Yaskawa INFORM job: FOLLOWBK.JBI

/JOB
//NAME FOLLOWBK
//POS
///NPOS 28,0,0,0,0,0
///TOOL 0
///POSTYPE PULSE
///PULSE
C00000=-2822,58859,-1118,-1041,-34109,-89
C00001=-2249,58669,-233,-1120,-33963,-317
C00002=-2249,58669,-1433,-1120,-33963,-317
C00003=-2021,58782,-1257,-1148,-34034,-410
C00004=-1683,58761,-1281,-1192,-34024,-546
C00005=-1595,58655,-1440,-1205,-33960,-580
C00006=-1505,58624,-1485,-1218,-33941,-615
C00007=-1505,58624,-285,-1218,-33941,-615
C00008=-1214,58456,-535,-1259,-33840,-730
C00009=-1214,58456,-1735,-1259,-33840,-730
C00010=-1059,58246,-2052,-1283,-33711,-789
C00011=-1059,58246,-852,-1283,-33711,-789
C00012=-2879,57741,-1646,-1051,-33397,-52
C00013=-2879,57741,-2846,-1051,-33397,-52
C00014=-2884,57537,-3152,-1053,-33275,-48
C00015=-2884,57537,-1952,-1053,-33275,-48
C00016=-2014,56709,-3199,-1183,-32765,-386
C00017=-2014,56709,-4399,-1183,-32765,-386
C00018=-1805,56927,-4068,-1207,-32897,-472
C00019=-1805,56927,-2868,-1207,-32897,-472
C00020=-1376,56655,-3280,-1270,-32726,-639
C00021=-1376,56655,-4480,-1270,-32726,-639
C00022=-1122,56919,-4076,-1299,-32888,-744
C00023=-1122,56919,-2876,-1299,-32888,-744
C00024=-2063,56484,-3540,-1180,-32628,-363
C00025=-2063,56484,-4740,-1180,-32628,-363
C00026=-1858,56475,-4754,-1208,-32620,-444
C00027=-1858,56475,-3554,-1208,-32620,-444
//INST
///DATE 2026/04/22 16:45
///ATTR SC,RW
///GROUP1 RB1
NOP
MOVJ C00000 VJ=0.78
MOVJ C00001 VJ=0.78
MOVJ C00002 VJ=0.78
MOVL C00003 V=12.0
MOVL C00004 V=12.0
MOVL C00005 V=12.0
MOVL C00006 V=12.0
MOVJ C00007 VJ=0.78
MOVJ C00008 VJ=0.78
MOVJ C00009 VJ=0.78
MOVL C00010 V=12.0
MOVJ C00011 VJ=0.78
MOVJ C00012 VJ=0.78
MOVJ C00013 VJ=0.78
MOVL C00014 V=12.0
MOVJ C00015 VJ=0.78
MOVJ C00016 VJ=0.78
MOVJ C00017 VJ=0.78
MOVL C00018 V=12.0
MOVJ C00019 VJ=0.78
MOVJ C00020 VJ=0.78
MOVJ C00021 VJ=0.78
MOVL C00022 V=12.0
MOVJ C00023 VJ=0.78
MOVJ C00024 VJ=0.78
MOVJ C00025 VJ=0.78
MOVL C00026 V=12.0
MOVJ C00027 VJ=0.78
END
